TYPE ST_LOG_EventData :
STRUCT
	bEnable					: BOOL;
	nCounter				: UDINT;
	sTimeStamp				: STRING;
	nImageByte				: UINT;
	aDataLogImage			: ARRAY[0..65000] OF BYTE;
	nMaxImageArraySize		: UINT := 65000 ;
	nControlSize			: UINT;
	bBufferOverflow			: BOOL;
END_STRUCT
END_TYPE

(* stored: Version 1.1.0.1
   DUT ST_LOG_EventData: Id {4463bd79-d049-4b66-ae3b-513f1a26e364} *)
